PROGRAM MAIN
VAR
	bLoad 	: BOOL;
	sPath	: STRING := 'C:\Temp\TC3_SyncUnits.pdf';
END_VAR

END_PROGRAM

(* stored: Version 1.1.0.1, ProductVersion 3.1.4024.3
   POU MAIN: Id {f4f0cafd-4cbb-483d-a3a6-3a1fa52891bd}, SpecialFunc None *)
